PROGRAM MAIN
VAR
END_VAR

END_PROGRAM

(* stored: Version 1.1.0.1
   POU MAIN: Id {581a0feb-1328-4d1d-92b6-fa21497d40e8} *)
